// TIA Portal V20 export
TYPE "LWONIK_typeFromSafetyDoorStatus"
// stored: Access Published
   STRUCT
      FdoorSwitchStatus { ExternalWritable := 'False'} : Struct
         anodeWasteDoorOpen : Bool;
         stackTableRearDoorOpen : Bool;
         cathodeWasteDoorOpen : Bool;
         unwinderRearDoorOpen : Bool;
         autoSpliceDoorOpen : Bool;
         unwinderMainDoorOpen : Bool;
         unwinderTopDoorOpen : Bool;
         unwinderBtmDoorOpen : Bool;
         StackTableDoorOpen : Bool;
         jrWinderDoorOpen : Bool;
      END_STRUCT;
      FdoorCoilStatus { ExternalWritable := 'False'} : Struct
         anodeWasteDoorUnlock : Bool;
         stackTableRearDoorUnlock : Bool;
         cathodeWasteDoorUnlock : Bool;
         unwinderRearDoorUnlock : Bool;
         autoSpliceDoorUnlock : Bool;
         unwinderMainDoorUnlock : Bool;
         unwinderTopDoorUnlock : Bool;
         unwinderBtmDoorUnlock : Bool;
         StackTableDoorUnlock : Bool;
         jrWinderDoorUnlock : Bool;
      END_STRUCT;
   END_STRUCT;
END_TYPE
